RoboDK station: HAMK_Robotics_station_MG400_with_camera.rdk

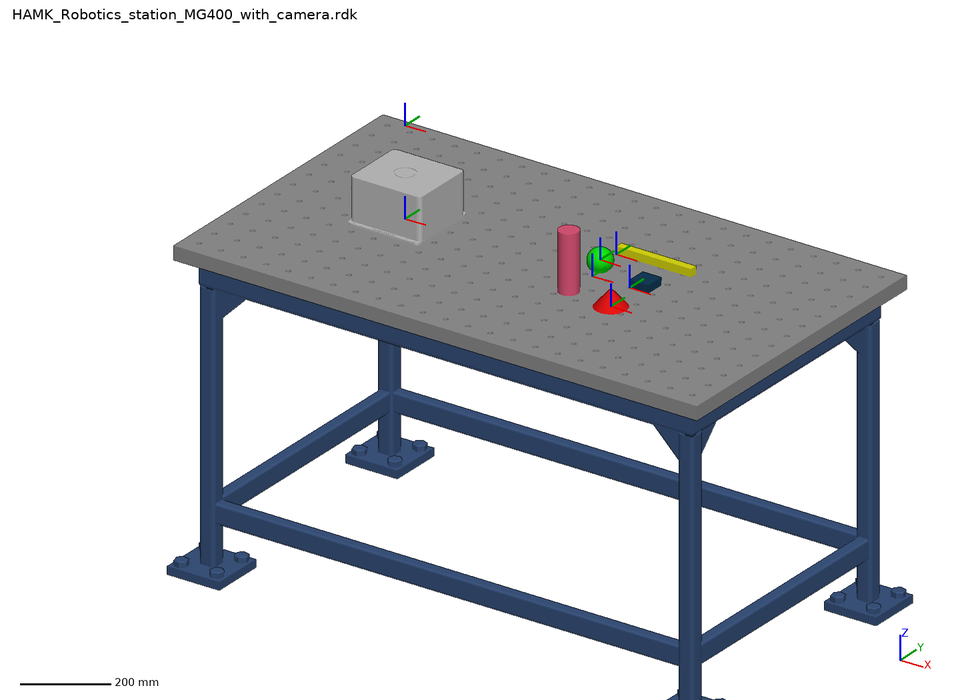
[picture v0: the station drawn from its stored meshes, robots at their saved joint values, targets as dots, program paths as lines]
Station HAMK_Robotics_station_MG400_with_camera (saved by RoboDK 5.9.4). Poses are relative to the parent item; angles as X-Y-Z fixed-axis rotations.
  - notes Note 1: <!DOCTYPE HTML PUBLIC "-//W3C//DTD HTML 4.0//EN" "http://www.w3.org/TR/REC-html40/strict.dtd">
<html><head><meta name="qrichtext" content="1" /><style type="text/css">
p, li { white-space: pre-wrap; }
</style></head><body style=" font-family:'MS Shell Dlg 2'; font-size:7.8pt; font-weight:400; font-style:normal;">
<p style=" margin-top:0px; margin-bottom:0px; margin-left:0px; margin-right:0px; -qt-block-indent:0; text-indent:0px;">In this station, a dummy tool (only the flange downloaded from https://uptimefab.com/2022/02/07/dobot-mg400/) is added to consider the 13mm of the tool shaft. Then, we use the coordinates of the TCP, that is, of the tip of the tool shaft.</p>
<p style=" margin-top:0px; margin-bottom:0px; margin-left:0px; margin-right:0px; -qt-block-indent:0; text-indent:0px;">Without any tool, the coordinates are refered to the robot flange.</p>
<p style=" margin-top:0px; margin-bottom:0px; margin-left:0px; margin-right:0px; -qt-block-indent:0; text-indent:0px;">Fernando S. Pacheco</p>
<p style=" margin-top:0px; margin-bottom:0px; margin-left:0px; margin-right:0px; -qt-block-indent:0; text-indent:0px;">September 2024</p>
<p style="-qt-paragraph-type:empty; margin-top:0px; margin-bottom:0px; margin-left:0px; margin-right:0px; -qt-block-indent:0; text-indent:0px;"><br /></p></body></html>
  - frame Dobot MG400 Base at (0, 0, 0) mm
    - robot Dobot MG400: 4 axes, payload 0.5 kg, reach 393.5 mm, repeatability 0.2 mm, weight 4 kg
        joint limits [-160, -25, -25, -360] to [160, 85, 105, 360]; home [0, 0, 0, 0]; saved at [0, 32.158, 32.645, 0]
      - tool MG400_End_Flange, TCP at (0, 0, -13) mm, size 39.8 x 39.8 x 14 mm
    - frame World at (0, 0, 0) mm
      - object Table 1400x800x800mm at (0, 0, 0) mm, size 1420 x 820 x 800 mm, geometry from Table-1400x800x800mm.sld
        - object HAMK logo at (360, 380, -115) mm, rotated rx 90 ry 0 rz 180 deg, size 301.4 x 100.9 x 9.4 mm, geometry from Fantastic Duup(2).stl
        - object white background at (360, 385.5, -110) mm, rotated rx 90 ry 0 rz 0 deg, size 480 x 184.8 x 2.4 mm, geometry from Fantastic Duup(3).stl
  - frame ReferenceFrameTCP at (0, 0, 227.75) mm
  - frame Camera Location Frame at (500, 0, 1000) mm, rotated rx 180 ry 0 rz -180 deg
  - frame Components at (500, 0, 0) mm
    - frame Box 1 at (100, 0, 0) mm
      - object Box 1 at (0, 0, 0) mm, size 50 x 50 x 20 mm, geometry from cube.sld
    - frame Sphere at (0, 30, 28) mm
      - object Sphere 1 at (0, 0, 0) mm, size 60 x 60 x 60 mm, geometry from sph.sld
    - frame Cone at (120, -100, 0) mm
      - object Cone 1 at (0, 0, 0) mm, size 80 x 80 x 40 mm
    - frame Box 2 at (-20, 120, 0) mm
      - object Box 1 at (0, 0, 0) mm, size 200 x 20 x 20 mm, geometry from cube.sld
  - object Cylinder 50x150mm at (500, -90, 0) mm, size 50 x 50 x 150 mm, geometry from Cylinder-50x150mm.sld
  - camera Camera 1
  - Python program Prog1 (listed below)

--- Python program Prog1 ---
from robodk import robolink

RDK = robolink.Robolink()

# Get camera object
cam = RDK.Item('Camera 1')  # Replace with your camera name

# Take a snapshot
success = cam.setParam('Open', 1)  # Open camera window

# Get and save image
file = RDK.getParam('PATH_OPENSTATION') + "/robodk_snapshot.png"
RDK.Cam2D_Snapshot(file, cam)
